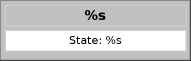
VISUALIZATION VFM_Module  // 191x61
VAR_IN_OUT
	HMI : ST_PackMLBaseModule_HMI;
END_VAR
    Rectangle (0,0 191x61)
    Textfield (5,5 181x21), "%s", text variable: HMI.Config.Name
    Textfield (5,30 181x21), "State: %s", text variable: HMI.Status.State
END_VISUALIZATION

(* stored: Version 1.1.0.1, ProductVersion 3.1.4024.12
   Visu VFM_Module: Id {c727be3e-f6ee-422a-a9fd-b0c3ffcb44f8} *)
